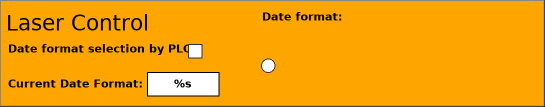
VISUALIZATION vLaserControl  // 545x107
VAR_IN_OUT
	stHMI: stHMI_Laser;
END_VAR
    Rectangle (0,0 545x107)
    RadioButton (259,32 150x67), variable: stHMI.iSelectMarking, input disabled if: GVL.fbUserLogin.nUserRole <> nSQL_UserRoles.Maintenance
        Areas[0]: Text=Year - Week
        Areas[1]: Text=Year - Month
    Label (5,37 226x24), "Date format selection by PLC"
    Label (9,63 226x24)
    Label (259,5 226x24), "Date format:"
    Checkbox (186,38 26x26), variable: stHMI.bEnableLaserTCPCOmmunication, input disabled if: GVL.fbUserLogin.nUserRole <> nSQL_UserRoles.Maintenance
    Label (5,72 226x24), "Current Date Format:"
    Rectangle (147,72 72x24), "%s", text variable: stHMI.sCurrentDateText, input disabled if: TRUE
    Label (3,8 156x30), "Laser Control"
END_VISUALIZATION

(* stored: Version 1.1.0.1, ProductVersion 3.1.4024.15
   Visu vLaserControl: Id {c08bbe31-27d0-4879-9423-9f1dc6b0888c} *)
